{attribute 'linkalways'} 
{attribute 'no_explicit_call' := 'This FB is a CLASS and must be accessed using methods or properties'}
{attribute 'enable_dynamic_creation'}
FUNCTION_BLOCK PendingResponseData EXTENDS Disposable IMPLEMENTS I_PendingResponseData
VAR
	_suggestedRetryDelayInMs : UDINT;
	state : (PENDING, SUCCESS, ERROR) := PENDING;
	errorMessage : T_MAXSTRING;
	pData : POINTER TO BYTE;
	dataSize : UDINT;
END_VAR

METHOD PUBLIC CopyPayloadData
VAR_INPUT
	PayloadDataAddress : PVOID;
	PayloadDataSize : UDINT;
END_VAR
dataSize := PayloadDataSize;
pData := __NEW(BYTE, PayloadDataSize);
memcpy(pData,PayloadDataAddress,PayloadDataSize);
END_METHOD

METHOD PRIVATE DeletePayloadData
VAR_INPUT
END_VAR
IF pData = 0 THEN
	RETURN;
END_IF

__DELETE(pData);
dataSize := 0;
END_METHOD

METHOD PUBLIC Error
VAR_INPUT
	Message : T_MAXSTRING;
END_VAR
IF state <> PENDING THEN
	RETURN;
END_IF

state := ERROR;
errorMessage := Message;
END_METHOD

METHOD FB_exit : BOOL
VAR_INPUT
	bInCopyCode : BOOL; // if TRUE, the exit method is called for exiting an instance that is copied afterwards (online change).
END_VAR
IF bInCopyCode THEN
	RETURN;
END_IF

DeletePayloadData();
END_METHOD

METHOD FB_init : BOOL
VAR_INPUT
	bInitRetains : BOOL; // if TRUE, the retain variables are initialized (warm start / cold start)
	bInCopyCode : BOOL;  // if TRUE, the instance afterwards gets moved into the copy code (online change)
	SuggestedRetryDelayInMs : UDINT;
END_VAR
_suggestedRetryDelayInMs := SuggestedRetryDelayInMs;
END_METHOD

PROPERTY PUBLIC IsPending : BOOL
GET
IsPending := state = PENDING;
END_GET
END_PROPERTY

METHOD PUBLIC Success
VAR_INPUT
	PayloadDataAddress : PVOID;
	PayloadDataSize : UDINT;
END_VAR
IF state <> PENDING THEN
	RETURN;
END_IF

state := SUCCESS;
CopyPayloadData(PayloadDataAddress, PayloadDataSize);
END_METHOD

PROPERTY PUBLIC SuggestedRetryDelayInMs : UDINT
GET
SuggestedRetryDelayInMs := _suggestedRetryDelayInMs;
END_GET
SET // PUBLIC
_suggestedRetryDelayInMs := SuggestedRetryDelayInMs;
END_SET
END_PROPERTY

METHOD PUBLIC TryUpdateServerResponse : BOOL
VAR_INPUT
	Response : I_ServerResponse;
END_VAR
IF state = ERROR THEN
	Response.Error(errorMessage);
	TryUpdateServerResponse := TRUE;
	RETURN;
END_IF

IF State = SUCCESS THEN
	Response.Success(pData,dataSize);
	TryUpdateServerResponse := TRUE;
	RETURN;
END_IF
END_METHOD

END_FUNCTION_BLOCK

(* stored: Version 1.1.0.1, ProductVersion 3.1.4024.12
   POU PendingResponseData: Id {e80c52bf-a657-4476-96bf-ac23d371397e}, SpecialFunc None
   Folder Constructor: Id {fd1d7c9c-8149-4e60-a630-ac53b72afc05}
   Folder Destructor: Id {92193c64-b8a1-4084-9f73-ede3cb9fc600}
   Folder Private: Id {7bfe6b87-3b8a-455d-86db-8158c4a2fdbd}
   Method CopyPayloadData: Id {e66372fa-7be6-4f89-8f8f-0a05a48e562f}
   Method DeletePayloadData: Id {598ea30b-cc57-4dd1-8279-3b57e55344fa}
   Method Error: Id {d8874e37-8230-4cfd-99a2-767b2709cfc7}
   Method FB_exit: Id {bd1bb881-c20d-4ede-87b1-508cc4ec0fb1}
   Method FB_init: Id {82a161ac-56ba-4700-8624-6ca1056a442f}
   Property IsPending: Id {73fe6f9a-3972-4114-b912-1cdd633f7015}
   Get Get: Id {35943817-8487-400b-adb0-f6d1f60328b7}
   Method Success: Id {ae814988-69a7-4780-8aa9-b373e08c0604}
   Property SuggestedRetryDelayInMs: Id {188e8b06-d5ec-41e3-81ef-1fe315326cab}
   Get Get: Id {ca2ed6f1-4b09-488e-adba-9274ce464b54}
   Set Set: Id {cd5cba61-bced-4f11-8bf0-1ca313739d04}
   Method TryUpdateServerResponse: Id {312b7c7f-0ca0-4541-b900-f6304201b4d3} *)
